TYPE E_Axis_C715 :
(
	E_C715_WALKINGBEAM	:=1,
	E_C715_ELEVATOR		:=2,
	E_C715_TRANSFER		:=3,
	E_C715_PRESENTATION	:=4

);
END_TYPE

(* stored: Version 1.1.0.1, ProductVersion 3.1.4024.15
   DUT E_Axis_C715: Id {f6c0327b-1e11-4ad0-b520-22f698317183} *)
